Omron CX-Programmer project НовыйПроект (CX-Programmer 9.61)

# PLC Svetofor: CP1L-E EM

## Global symbols (name address type ; comment)
100.04 BOOL  ; кр п
T0000 BOOL  ; красный
T0001 BOOL  ; красный + желтый
T0002 BOOL  ; зеленый
T0003 BOOL  ; зеленый мигающий
T0004 BOOL  ; красн п
T0005 BOOL  ; желтый вкл
T0006 BOOL  ; желтый выкл
T0007 BOOL  ; зеленый вкл
T0008 BOOL  ; зеленый выкл
W5 CHANNEL  ; Время * 10
Time W1 UINT  ; Время фазы
Visible W0.00 BOOL  ; Отображение времени
green 100.02 BOOL  ; зеленый
red 100.00 BOOL  ; красный
run 0.00 BOOL  ; работа
t_green H1 UINT  ; время зеленого 0,1с
t_red H0 UINT  ; время красного 0,1с
yellow 100.01 BOOL  ; желтый

## Program НоваяЗадача1 (cyclic task 0)

### Section Сегмент1

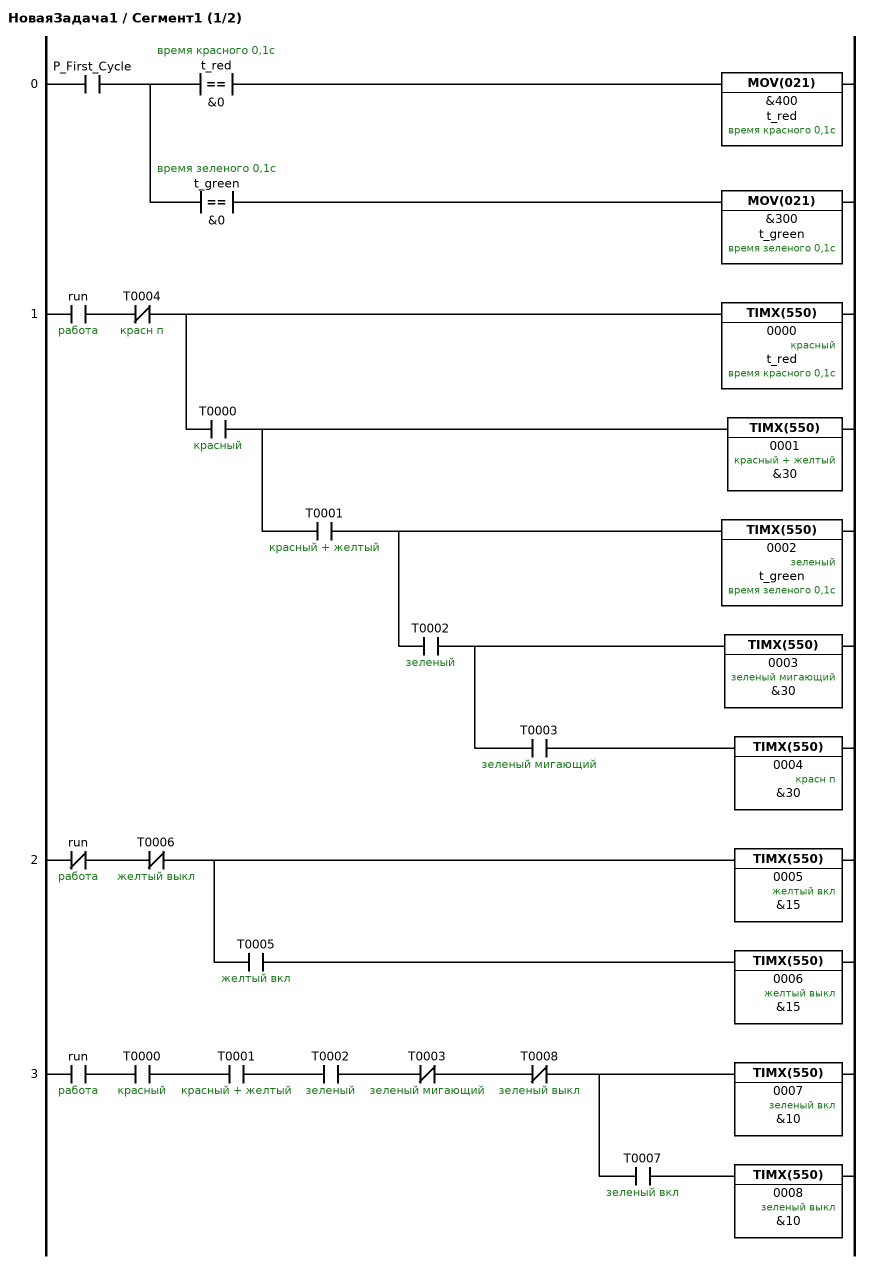
; rung 0
LD P_First_Cycle
OUT TR0
AND=(300) t_red &0  ; время красного 0,1с
MOV(021) &400 t_red  ; время красного 0,1с
LD TR0
AND=(300) t_green &0  ; время зеленого 0,1с
MOV(021) &300 t_green  ; время зеленого 0,1с
; rung 1
LD run  ; работа
ANDNOT T0004  ; красн п
TIMX(550) 0000 t_red  ; время красного 0,1с, красный
AND T0000  ; красный
TIMX(550) 0001 &30  ; красный + желтый
AND T0001  ; красный + желтый
TIMX(550) 0002 t_green  ; время зеленого 0,1с, зеленый
AND T0002  ; зеленый
TIMX(550) 0003 &30  ; зеленый мигающий
AND T0003  ; зеленый мигающий
TIMX(550) 0004 &30  ; красн п
; rung 2
LDNOT run  ; работа
ANDNOT T0006  ; желтый выкл
TIMX(550) 0005 &15  ; желтый вкл
AND T0005  ; желтый вкл
TIMX(550) 0006 &15  ; желтый выкл
; rung 3
LD run  ; работа
AND T0000  ; красный
AND T0001  ; красный + желтый
AND T0002  ; зеленый
ANDNOT T0003  ; зеленый мигающий
ANDNOT T0008  ; зеленый выкл
TIMX(550) 0007 &10  ; зеленый вкл
AND T0007  ; зеленый вкл
TIMX(550) 0008 &10  ; зеленый выкл

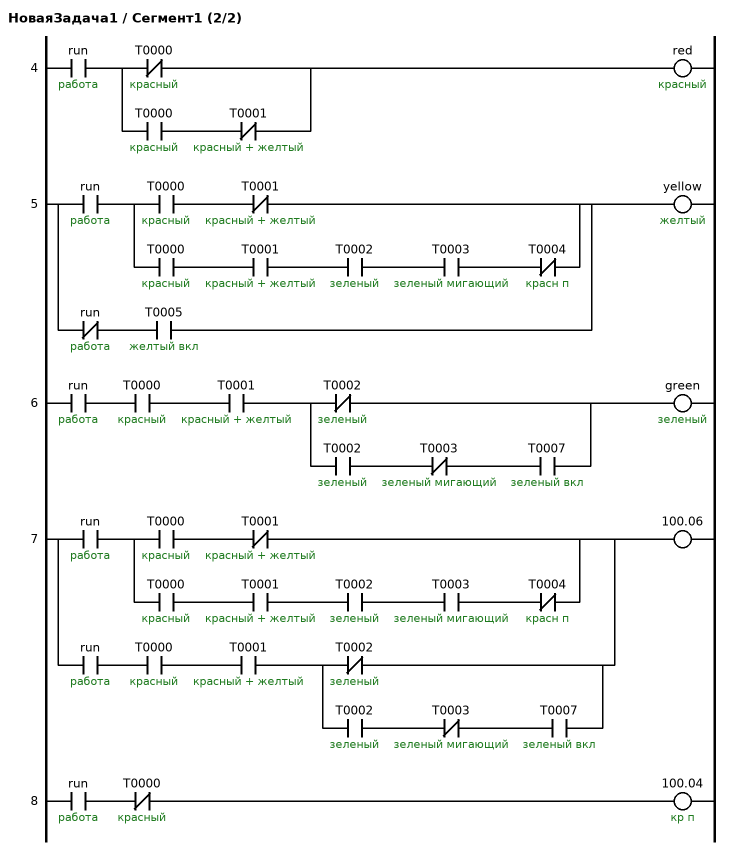
; rung 4
LD run  ; работа
LDNOT T0000  ; красный
LD T0000  ; красный
ANDNOT T0001  ; красный + желтый
ORLD
ANDLD
OUT red  ; красный
; rung 5
LD run  ; работа
LD T0000  ; красный
ANDNOT T0001  ; красный + желтый
LD T0000  ; красный
AND T0001  ; красный + желтый
AND T0002  ; зеленый
AND T0003  ; зеленый мигающий
ANDNOT T0004  ; красн п
ORLD
ANDLD
LDNOT run  ; работа
AND T0005  ; желтый вкл
ORLD
OUT yellow  ; желтый
; rung 6
LD run  ; работа
AND T0000  ; красный
AND T0001  ; красный + желтый
LDNOT T0002  ; зеленый
LD T0002  ; зеленый
ANDNOT T0003  ; зеленый мигающий
AND T0007  ; зеленый вкл
ORLD
ANDLD
OUT green  ; зеленый
; rung 7
LD run  ; работа
LD T0000  ; красный
ANDNOT T0001  ; красный + желтый
LD T0000  ; красный
AND T0001  ; красный + желтый
AND T0002  ; зеленый
AND T0003  ; зеленый мигающий
ANDNOT T0004  ; красн п
ORLD
ANDLD
LD run  ; работа
AND T0000  ; красный
AND T0001  ; красный + желтый
LDNOT T0002  ; зеленый
LD T0002  ; зеленый
ANDNOT T0003  ; зеленый мигающий
AND T0007  ; зеленый вкл
ORLD
ANDLD
ORLD
OUT 100.06
; rung 8
LD run  ; работа
ANDNOT T0000  ; красный
OUT 100.04  ; кр п

### Section Сегмент2

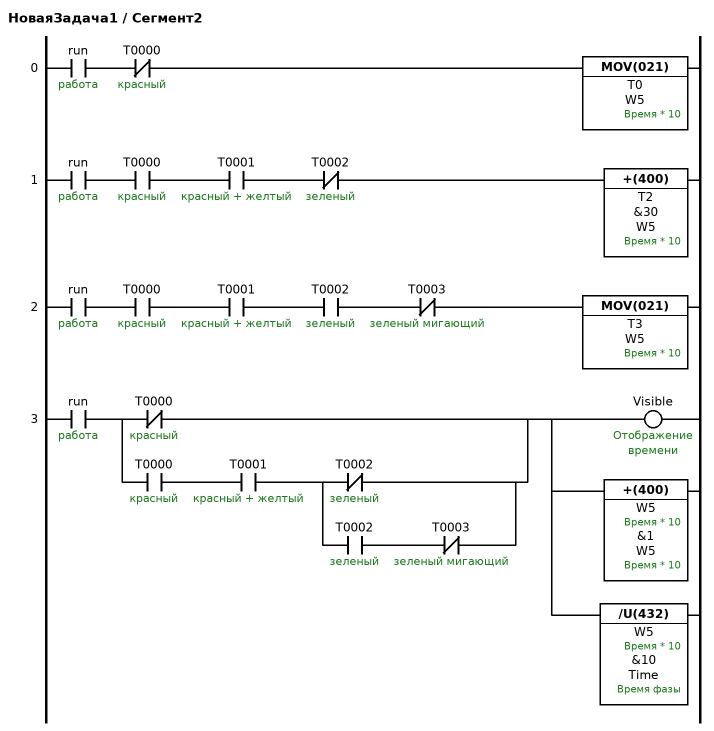
; rung 0
LD run  ; работа
ANDNOT T0000  ; красный
MOV(021) T0 W5  ; Время * 10
; rung 1
LD run  ; работа
AND T0000  ; красный
AND T0001  ; красный + желтый
ANDNOT T0002  ; зеленый
+(400) T2 &30 W5  ; Время * 10
; rung 2
LD run  ; работа
AND T0000  ; красный
AND T0001  ; красный + желтый
AND T0002  ; зеленый
ANDNOT T0003  ; зеленый мигающий
MOV(021) T3 W5  ; Время * 10
; rung 3
LD run  ; работа
LDNOT T0000  ; красный
LD T0000  ; красный
AND T0001  ; красный + желтый
LDNOT T0002  ; зеленый
LD T0002  ; зеленый
ANDNOT T0003  ; зеленый мигающий
ORLD
ANDLD
ORLD
ANDLD
OUT Visible  ; Отображение времени
+(400) W5 &1 W5  ; Время * 10
/U(432) W5 &10 Time  ; Время * 10, Время фазы

### Section END
; rung 0
END(001)